// TwinCAT 3 PLC project MotionDevicesPackage
// ProgramVersion: 3.1.4023.0
// libraries:
//   Tc2_MC2, * (Beckhoff Automation GmbH)
//   Tc2_Standard, * (Beckhoff Automation GmbH)
//   Tc2_System, * (Beckhoff Automation GmbH)
//   Tc3_Module, * (Beckhoff Automation GmbH)
// project tree:
//   DUTs/Conveyors/ Conveyor.TcPOU (not stored), ConveyorLSC.TcPOU, ConveyorMode.TcDUT, ConveyorSC.TcPOU, ConveyorSC_NC.TcPOU
//   DUTs/Insertion Package/Drives/ AirPiston.TcPOU, ClearLinkMC.TcPOU, ServoNC.TcPOU, SimplePiston.TcPOU
//   DUTs/Insertion Package/ Homing.TcDUT, Insertion.TcPOU, SuctionPad.TcDUT (not stored)
//   DUTs/Insertion Package/Prototypes/ FBA_Drive.TcPOU, FBA_TrifectaDrive.TcPOU, I_ContinuousDrive.TcIO, I_Drive.TcIO, I_EncodedDrive.TcIO, I_PositionalDrive.TcIO
//   / PlcTask3.TcTTO
//   POUs/ MAIN.TcPOU, WithinTolerance.TcPOU
// (motion and I/O tree: see PLC project conveyorslinking)
// real-time tasks:
//   TASK PlcTask: cycle T#10ms, priority 20, ADS port 350
//   TASK PlcTask1: cycle T#10ms, priority 21, ADS port 351
//   TASK PlcTask2: cycle T#10ms, priority 22, ADS port 352
//   TASK PlcTask3: cycle T#10ms, priority 23, ADS port 353

CONFIGURATION MotionDevicesPackage
    RESOURCE PLC ON TwinCAT3
        TASK PlcTask3(INTERVAL := T#10ms, PRIORITY := 23);
        PROGRAM MAIN WITH PlcTask3 : MAIN;
    END_RESOURCE
END_CONFIGURATION

// ---- DUTs/Conveyors/ConveyorMode.TcDUT
{attribute 'qualified_only'}
//{attribute 'strict'}
TYPE ConveyorMode :
(
	IDLE,
	FORWARD,
	BACKWARD,
	STOP,
	
	size
);
END_TYPE

// ---- DUTs/Insertion Package/Homing.TcDUT
{attribute 'qualified_only'}
{attribute 'strict'}
TYPE Homing :
(
	IDLE,
	
	START,
	RETRY,
	
	STOP,
	SET,
	DONE,
	
	size
);
END_TYPE
(*
general homing sequence:
	on drive.homingSequence() call, home towards home sensor
	if home reached, set position and finish homing as usual
	if outer limit reached, traverse towards inner limit
		when inner limit reached, retry homing
*)

// ---- DUTs/Insertion Package/Prototypes/I_ContinuousDrive.TcIO
INTERFACE I_ContinuousDrive EXTENDS I_Drive

METHOD ABSTRACT moveContinuous : BOOL
VAR_INPUT
	direction : MC_Direction;
END_VAR
END_METHOD

END_INTERFACE

// ---- DUTs/Insertion Package/Prototypes/I_Drive.TcIO
INTERFACE I_Drive

{attribute 'monitoring':='call'}
PROPERTY Active : BOOL
GET
END_GET
END_PROPERTY

{attribute 'monitoring':='call'}
PROPERTY AtHome : BOOL
GET
END_GET
END_PROPERTY

{attribute 'monitoring':='call'}
PROPERTY Error : BOOL
GET
END_GET
END_PROPERTY

{attribute 'monitoring':='call'}
PROPERTY HomeSet : BOOL
GET
END_GET
END_PROPERTY

METHOD ABSTRACT homingSequence : BOOL
VAR_INPUT
END_VAR
END_METHOD

METHOD reset : BOOL
VAR_INPUT
END_VAR
END_METHOD

METHOD ABSTRACT stop : BOOL
VAR_INPUT
END_VAR
END_METHOD

METHOD toHome : BOOL
VAR_INPUT
END_VAR
END_METHOD

END_INTERFACE

// ---- DUTs/Insertion Package/Prototypes/I_EncodedDrive.TcIO
INTERFACE I_EncodedDrive EXTENDS I_PositionalDrive, I_ContinuousDrive
//this drive can perform absolute/relative targeting and continuous motion
//only used if a drive with both encoded and continuous behavior is needed

END_INTERFACE

// ---- DUTs/Insertion Package/Prototypes/I_PositionalDrive.TcIO
INTERFACE I_PositionalDrive EXTENDS I_Drive

PROPERTY CurrentPosition : LREAL
GET
END_GET
SET
END_SET
END_PROPERTY

METHOD ABSTRACT moveAbsolute : BOOL
VAR_INPUT
	newTarget : LREAL; 
END_VAR
END_METHOD

METHOD ABSTRACT moveRelative : BOOL
VAR_INPUT
	distance : LREAL;
END_VAR
END_METHOD

PROPERTY TargetPosition : LREAL
GET
END_GET
SET
END_SET
END_PROPERTY

END_INTERFACE

// ---- POUs/MAIN.TcPOU
PROGRAM MAIN
VAR
	xInsertion : Insertion;
	
	xServoNC : ServoNC;
	xClearLinkMC : ClearLinkMC;
	xAirPiston : AirPiston;
	xSimplePiston : SimplePiston;
	
	xConveyorSC : ConveyorSC;
	xConveyorLSC : ConveyorLSC;
	xConveyorSC_NC : ConveyorSC_NC;
END_VAR

(*
this solution contains the package for various motion devices and the inheritance hierarchy, and any additional types
the Insertion Package folder under DUTs + WithinTolerance() can be copied to any project/module as needed

I_Drive contains the minimum behavior for any drive
FBA_Drive implements I_Drive with the minimum declaration
	FBA_TrifectaDrive extends it by adding an outer limit sensor for drives requiring 3 sensors
	
all Insertion-capable drives extend FBA_Drive or FBA_TrifectaDrive and implement I_ContinuousDrive, I_PositionalDrive, or I_EncodedDrive
*)

END_PROGRAM

// ---- DUTs/Insertion Package/Insertion.TcPOU
FUNCTION_BLOCK Insertion //2d insertion that combines a slider (alignment) and screw (push)
VAR_INPUT //interface references to existing drives
	slider : I_PositionalDrive;
	screw : I_ContinuousDrive;
END_VAR
VAR_OUTPUT
	contact AT %I* : BOOL;
	
	active : BOOL;
	error : BOOL;
	home : BOOL;
	
	homingComplete : BOOL;
	
	sliderPos : LREAL;
END_VAR
(*
this FB encapsulates 2 drives into a generic insertion machine
both drives should be declared externally in Hardware GVL as a concrete FB
Insertion instance should be declared and called in module scope, with the drives from Hardware GVL passed in by Interface reference
*)

homingComplete := slider.HomeSet AND screw.HomeSet;

active := slider.Active OR screw.Active;
error := slider.Error OR screw.Error;
home := slider.AtHome AND screw.AtHome;

sliderPos := slider.CurrentPosition;

METHOD align : BOOL
VAR_INPUT
	targetPos : REAL;
END_VAR
slider.moveAbsolute(newTarget := targetPos);
END_METHOD

METHOD homingSequence : BOOL
VAR_INPUT
END_VAR
IF NOT slider.homeSet THEN
	slider.homingSequence();
END_IF

IF NOT screw.homeSet THEN
	screw.homingSequence();
END_IF

homingSequence := homingComplete;
END_METHOD

METHOD press : BOOL
VAR_INPUT
END_VAR
IF NOT contact THEN
	screw.moveContinuous(direction := MC_Negative_Direction);
END_IF
END_METHOD

METHOD release : BOOL
VAR_INPUT
END_VAR
screw.moveContinuous(direction := MC_Positive_Direction);
END_METHOD

METHOD reset : BOOL
VAR_INPUT
END_VAR
slider.reset();
screw.reset();
END_METHOD

METHOD stop : BOOL
VAR_INPUT
END_VAR
screw.stop();
slider.stop();
END_METHOD

METHOD toHome : BOOL
VAR_INPUT
END_VAR
slider.toHome();
screw.toHome();

toHome := slider.AtHome AND screw.AtHome;
END_METHOD

END_FUNCTION_BLOCK

// ---- DUTs/Insertion Package/Drives/ServoNC.TcPOU
FUNCTION_BLOCK ServoNC EXTENDS FBA_TrifectaDrive IMPLEMENTS I_EncodedDrive
VAR_OUTPUT	
	ready : BOOL;
	position : LREAL;
	velocity : LREAL;
END_VAR
VAR
	axis : AXIS_REF;
	
	mcReadPosition : MC_ReadActualPosition; //continuous enable FBs
	mcReadVelocity : MC_ReadActualVelocity;
	mcReadError : MC_ReadAxisError;
	mcPower : MC_Power;
	
	mcReset : MC_Reset; //rising edge FBs
	mcMoveAbsolute : MC_MoveAbsolute;
	mcMoveRelative : MC_MoveRelative;
	mcMoveVelocity : MC_MoveVelocity;
	
	mcSetPosition : MC_SetPosition;
	mcStop : MC_Stop;
END_VAR
VAR_STAT CONSTANT
	targetingVelocity : INT := 500;
	continuousVelocity : INT := 100;
END_VAR

override();

blocks();

mcReset.Execute := FALSE;
mcMoveAbsolute.Execute := FALSE;
mcMoveRelative.Execute := FALSE;
mcMoveVelocity.Execute := FALSE;
mcSetPosition.Execute := FALSE;
mcStop.Execute := FALSE;

blocks();

ready := bEnable AND NOT Active AND HomeSet;

PROPERTY Active : BOOL
GET
Active := 
	mcMoveAbsolute.Busy OR 
	mcMoveRelative.Busy OR 
	mcMoveVelocity.Busy OR 
	mcSetPosition.Busy OR 
	mcReset.Busy OR 
	mcStop.Busy OR 
	step <> 0;
END_GET
END_PROPERTY

METHOD PRIVATE blocks : BOOL
mcReadPosition(
	Axis:= axis, 
	Enable:= TRUE, 
	Valid=> , 
	Busy=> , 
	Error=> , 
	ErrorID=> , 
	Position=> position);
	
mcReadVelocity(
	Axis:= axis, 
	Enable:= TRUE, 
	Valid=> , 
	Busy=> , 
	Error=> , 
	ErrorID=> , 
	ActualVelocity=> velocity);
	
mcReadError(
	Axis:= axis, 
	Enable:= TRUE, 
	Valid=> , 
	Busy=> , 
	Error=> , 
	ErrorID=> , 
	AxisErrorID=> );

mcReset(
	Axis:= axis, 
	Execute:= , 
	Done=> , 
	Busy=> , 
	Error=> , 
	ErrorID=> );

mcPower(
	Axis:= axis, 
	Enable:= bEnable, 
	Enable_Positive:= TRUE, 
	Enable_Negative:= TRUE, 
	Override:= 100, 
	BufferMode:= , 
	Options:= , 
	Status=> , 
	Busy=> , 
	Active=> , 
	Error=> , 
	ErrorID=> );

mcMoveAbsolute(
	Axis:= axis, 
	Execute:= , 
	Position:= , 
	Velocity:= targetingVelocity, 
	Acceleration:= , 
	Deceleration:= , 
	Jerk:= , 
	BufferMode:= , 
	Options:= , 
	Done=> , 
	Busy=> , 
	Active=> , 
	CommandAborted=> , 
	Error=> , 
	ErrorID=> );
	
mcMoveRelative(
	Axis:= axis, 
	Execute:= , 
	Distance:= ,
	Velocity:= targetingVelocity, 
	Acceleration:= , 
	Deceleration:= , 
	Jerk:= , 
	BufferMode:= , 
	Options:= , 
	Done=> , 
	Busy=> , 
	Active=> , 
	CommandAborted=> , 
	Error=> , 
	ErrorID=> );
	
mcMoveVelocity( //stopped with stop();
	Axis:= axis, 
	Execute:= , 
	Velocity:= continuousVelocity, 
	Acceleration:= , 
	Deceleration:= , 
	Jerk:= , 
	Direction:= , 
	BufferMode:= , 
	Options:= , 
	InVelocity=> , 
	Busy=> , 
	Active=> , 
	CommandAborted=> , 
	Error=> , 
	ErrorID=> );
	
mcSetPosition(
	Axis:= axis, 
	Execute:= , 
	Position:= , 
	Mode:= , 
	Options:= , 
	Done=> , 
	Busy=> , 
	Error=> , 
	ErrorID=> );
	
mcStop(
	Axis:= axis, 
	Execute:= , 
	Deceleration:= , 
	Jerk:= , 
	Options:= , 
	Done=> , 
	Busy=> , 
	Active=> , 
	CommandAborted=> , 
	Error=> , 
	ErrorID=> );
END_METHOD

PROPERTY CurrentPosition : LREAL
GET
CurrentPosition := position;
END_GET
SET
position := CurrentPosition;
END_SET
END_PROPERTY

PROPERTY Error : BOOL
GET
error := 
	mcMoveAbsolute.Error OR 
	mcMoveRelative.Error OR 
	mcMoveVelocity.Error OR 
	mcSetPosition.Error OR 
	mcReset.Error OR 
	mcStop.Error OR
	mcReadError.AxisErrorID > 0;
END_GET
END_PROPERTY

METHOD homingSequence : BOOL
CASE step OF
	Homing.IDLE:
		reset();
		IF bEnable THEN
			step := Homing.START;
		END_IF
		
	Homing.START:
		IF AtHome THEN
			mcMoveVelocity.Execute := FALSE;
			step := Homing.STOP;
			
		ELSIF AtInnerLimit THEN
			mcMoveVelocity.Execute := FALSE;
			step := Homing.RETRY;
			
		ELSE
			mcMoveVelocity.Direction := MC_Negative_Direction;
			mcMoveVelocity.Execute := NOT mcMoveVelocity.Execute;
		END_IF
		
	Homing.RETRY:
		IF AtOuterLimit THEN
			mcMoveVelocity.Execute := FALSE;
			step := Homing.START;
		ELSE
			mcMoveVelocity.Direction := MC_Positive_Direction;
			mcMoveVelocity.Execute := NOT mcMoveVelocity.Execute;
		END_IF
		
	Homing.STOP:
		IF velocity = 0 THEN
			mcStop.Execute := FALSE;
			step := Homing.SET;
		ELSE
			mcStop.Execute := TRUE;
		END_IF
		
	Homing.SET:
		IF position = 0 THEN
			mcSetPosition.Execute := FALSE;
			homingSequence := TRUE;
			step := Homing.DONE;
		ELSE
			mcSetPosition.Position := 0;
			mcSetPosition.Execute := TRUE;
		END_IF
		
	Homing.DONE:
		homingComplete := TRUE;
		step := Homing.IDLE;
		
END_CASE
END_METHOD

METHOD moveAbsolute : BOOL
VAR_INPUT
	newTarget : LREAL;
END_VAR
(*
VAR_OUTPUT
	fault : BOOL;
END_VAR
*)
IF NOT Active AND NOT error THEN
	mcMoveAbsolute.Position := newTarget;
	mcMoveAbsolute.Execute := TRUE;
END_IF

moveAbsolute := (*mcMoveAbsolute.Done AND mcMoveAbsolute.Active;*)
	position = newTarget;
END_METHOD

METHOD moveContinuous : BOOL
VAR_INPUT
	//direction : BOOL; //direction (F = inwards, T = outwards)
	direction : MC_Direction;
END_VAR
(*
IF mcMoveVelocity.Active THEN
	stop();
END_IF

IF NOT mcStop.Done THEN
	RETURN;
END_IF
*)
(*
IF direction THEN
	mcMoveVelocity.Direction := MC_Positive_Direction;
ELSE
	mcMoveVelocity.Direction := MC_Negative_Direction;
END_IF
*)
mcMoveVelocity.Direction := direction;

IF NOT mcMoveVelocity.Error THEN
	mcMoveVelocity.Execute := TRUE;
	moveContinuous := TRUE;
END_IF
END_METHOD

METHOD moveRelative : BOOL
VAR_INPUT
	distance : LREAL;
END_VAR
mcMoveRelative.Distance := distance;

moveRelative := mcMoveRelative.Done;
END_METHOD

METHOD PRIVATE override : BOOL
VAR_INPUT
END_VAR
(*
-at home and attempting to traverse outward
-at outer limit and attempting to traverse outward
-at inner limit and attempting to traverse inwards
*)
(*
inward = negative direction, negative velocity
outward = positive direction, positive velocity
*)

IF error THEN
	stop();
	reset();
	
ELSIF
	AtHome AND (TargetPosition > CurrentPosition OR velocity > 0) OR
	AtInnerLimit AND (TargetPosition > CurrentPosition OR velocity > 0) OR
	AtOuterLimit AND (TargetPosition < CurrentPosition OR velocity < 0)
THEN
	stop();
END_IF
END_METHOD

METHOD reset : BOOL
VAR_INPUT
END_VAR
mcReset.Execute := TRUE;

reset := mcReset.Done;
END_METHOD

METHOD stop : BOOL
VAR_INPUT
END_VAR
mcStop.Execute := TRUE;

mcMoveAbsolute.Execute := FALSE;
mcMoveRelative.Execute := FALSE;
mcMoveVelocity.Execute := FALSE;
END_METHOD

PROPERTY TargetPosition : LREAL
GET
END_GET
SET
moveAbsolute(newTarget := TargetPosition);
END_SET
END_PROPERTY

METHOD toHome : BOOL
VAR_INPUT
END_VAR
moveAbsolute(newTarget := 0);

toHome := AtHome;
END_METHOD

END_FUNCTION_BLOCK

// ---- DUTs/Insertion Package/Prototypes/FBA_TrifectaDrive.TcPOU
FUNCTION_BLOCK ABSTRACT FBA_TrifectaDrive EXTENDS FBA_Drive
VAR
	outerLimit AT %I* : BOOL;
END_VAR
(*
this abstract FB adds a rear limit sensor to FBA_Drive
*)

{attribute 'monitoring':='call'}
PROPERTY AtOuterLimit : BOOL
GET
AtOuterLimit := outerLimit <> limitSensorDefaultState;
END_GET
END_PROPERTY

END_FUNCTION_BLOCK

// ---- DUTs/Insertion Package/Prototypes/FBA_Drive.TcPOU
FUNCTION_BLOCK ABSTRACT FBA_Drive IMPLEMENTS I_Drive
VAR_INPUT
	bEnable : BOOL;
END_VAR
VAR //constructor
	limitSensorDefaultState : BOOL;
	//when a traverse sensor is opposite of this value, the respective property becomes TRUE
	//all sensors for a drive should be of the same type - do not mix & match PNP and NPN sensors on the same drive
END_VAR
VAR		
	homingComplete : BOOL;
	step : Homing;
	
	innerLimit AT %I* : BOOL; //replacable with homeLimit
	home AT %I* : BOOL;
	//not all drives have a rear limit, drives that do must extend from FBA_TrifectaDrive
END_VAR
(*
this abstract FB only specifies the minimum data for any drive
*)

{attribute 'monitoring':='call'}
PROPERTY ABSTRACT Active : BOOL
GET
END_GET
END_PROPERTY

{attribute 'monitoring':='call'}
PROPERTY AtHome : BOOL
GET
AtHome := home <> limitSensorDefaultState;
END_GET
END_PROPERTY

{attribute 'monitoring':='call'}
PROPERTY AtInnerLimit : BOOL
GET
AtInnerLimit := innerLimit <> limitSensorDefaultState;
END_GET
END_PROPERTY

{attribute 'monitoring':='call'}
PROPERTY ABSTRACT Error : BOOL
GET
END_GET
END_PROPERTY

{attribute 'monitoring':='call'}
PROPERTY HomeSet : BOOL
GET
HomeSet := homingComplete;
END_GET
END_PROPERTY

{attribute 'TcRpcEnable'}
METHOD ABSTRACT homingSequence : BOOL
VAR_INPUT
END_VAR
END_METHOD

{attribute 'TcRpcEnable'}
METHOD ABSTRACT reset : BOOL
VAR_INPUT
END_VAR
END_METHOD

{attribute 'TcRpcEnable'}
METHOD ABSTRACT stop : BOOL
VAR_INPUT
END_VAR
END_METHOD

METHOD ABSTRACT toHome : BOOL
VAR_INPUT
END_VAR
END_METHOD

END_FUNCTION_BLOCK

// ---- DUTs/Insertion Package/Drives/ClearLinkMC.TcPOU
FUNCTION_BLOCK ClearLinkMC EXTENDS FBA_TrifectaDrive IMPLEMENTS I_EncodedDrive
VAR_OUTPUT
	pulse AT %Q* : INT;
	brakeRelease AT %Q* : BOOL := TRUE;
	enable : BOOL;
	A : BOOL;
	B : BOOL;
	clear : BOOL;
END_VAR
VAR	
	hlfb AT %I* : REAL := -9999; //high level feedback, if -9999 then servo is idle
	
	outputRegister AT %Q* : INT;
	pulseRequest : INT;
	
	homingDelay : TON;
	resetPulse : TP;
	
	mode : (HOLD, TARGET, CONTINUOUS, RESET_ERR);
	calculation : (IDLE, DOWN, UP, CALCULATE, DONE);
	maxPosition : LREAL;
	
	position, targetPos : LREAL;
	
	pulsePosition : INT;
	pulseCounter : INT;
	rotationsPerPulse : INT; //revolutions per pulse
	displacementPerPulse : LREAL; //displacement per pulse
END_VAR
VAR_STAT CONSTANT
	resetWidth : TIME := T#500MS;
	delayWidth : TIME := T#500MS;
END_VAR
VAR //constructor
	homingDirectionOut : BOOL; 			//homing direction - see <A>
	minPosition : LREAL;
	displacementPerRotation : LREAL; 	//displacement per revolution	
	unitsPerPulse : INT := 800; 		//800 Teknic units per rotation - default setting is 800 units (1 rotation) per pulse
END_VAR

//M-connector output register
outputRegister.0 := enable AND bEnable; 	//enable
outputRegister.1 := A; 						//direction bit - T = outwards, F = inwards
outputRegister.2 := B; 						//homing bit - after startup, set to TRUE to begin homing, then set to FALSE to finish homing
outputRegister.3 := clear; 					//reset bit

rotationsPerPulse := unitsPerPulse/800; //Teknic constant - 800 units per rotation
displacementPerPulse := displacementPerRotation * rotationsPerPulse;

resetPulse(IN:= , PT:= resetWidth, Q=> clear, ET=> ); //reset pulse

IF NOT enable AND NOT AtInnerLimit THEN
	homingComplete := FALSE;
	step := Homing.IDLE;
	mode := HOLD;
END_IF

override();

CASE mode OF		
	HOLD: //hold current position, no motion
		pulse := 0;
		pulseRequest := 0;
	
	TARGET:	//target a given position
		
		IF WithinTolerance(position, targetPos, displacementPerPulse) THEN
			pulseRequest := 0;
			pulse := 0;
			mode := HOLD;
			
		ELSIF NOT Active THEN
			A :=  position < targetPos;
			(*
			2 options to traverse to a target position:
				a)  send all pulses at once - continuous motion but may exceed limits, check for bounds before setting
				b)  1 pulse at a time - choppy but safer
			*)
			targetPos := MAX(targetPos, minPosition); //if below minPosition, set to minPosition
			targetPos := MIN(targetPos, maxPosition); //if above maxPosition, set to maxPosition
			
			pulseRequest := TO_INT(ABS(position - targetPos)/displacementPerPulse);
			//pulseRequest := 1;
		END_IF
		
	CONTINUOUS: //single pulses in the direction specified by moveContinuous()
		pulseRequest := 1;
		
	RESET_ERR: //reset pulse, servo may need to be rehomed aftewards
		pulse := 0;
		pulseRequest := 0;
		resetPulse.IN := TRUE;
		
		IF resetPulse.Q THEN
			resetPulse.IN := FALSE;
			mode := HOLD;
		END_IF
		
END_CASE

sequence();

PROPERTY Active : BOOL
GET
Active := hlfb <> -9999;
END_GET
END_PROPERTY

{attribute 'monitoring':='call'}
PROPERTY AtOuterLimit : BOOL
GET
AtOuterLimit := outerLimit <> limitSensorDefaultState;
END_GET
END_PROPERTY

METHOD PRIVATE calculatePositions : BOOL
(*
the purpose of this method is calculate the position at the outer limit

complete a full range traverse while counting the pulses, then multiply
	displacement per rotation
	rotations per pulse
	number of pulses for the traversal
and add to position at inner limit to get position at outer limit
*)
CASE calculation OF
	IDLE:
		calculation := DOWN;
		
	DOWN:
		moveContinuous(direction := MC_Negative_Direction);
		IF AtInnerLimit THEN
			calculation := UP;
			pulseCounter := 0;
		END_IF
		
	UP:
		moveContinuous(direction := MC_Positive_Direction);
		IF AtHome THEN
			maxPosition := minPosition + (displacementPerRotation * rotationsPerPulse * pulseCounter);
			calculation := DONE;
		END_IF
		
	DONE:
		calculation := 0;
		calculatePositions := TRUE;
		
END_CASE
END_METHOD

PROPERTY CurrentPosition : LREAL
GET
CurrentPosition := position;

//CurrentPosition := pulsePosition * displacementPerPulse;
END_GET
SET
position := CurrentPosition;
END_SET
END_PROPERTY

PROPERTY Error : BOOL
GET
END_GET
END_PROPERTY

METHOD homingSequence : BOOL
homingDelay(IN:= , PT:= delayWidth, Q=> , ET=> );

CASE step OF
	Homing.IDLE:
		enable := TRUE;
		A := FALSE;
		B := TRUE;
		brakeRelease := TRUE;
		
		homingComplete := FALSE;
		
		homingDelay.IN := TRUE;
		IF homingDelay.Q THEN
			homingDelay.IN := FALSE;
			//step := Homing.START;
			step := Homing.RETRY;
		END_IF
		
	Homing.START:
		IF homingDelay.Q THEN
			homingDelay.IN := FALSE;
			step := Homing.SET;
			
		ELSIF AtHome THEN
			homingDelay.IN := TRUE;
			
		ELSIF AtOuterLimit THEN
			step := Homing.RETRY;
		
		ELSE
			enable := TRUE;
			A := FALSE;
			B := TRUE;
			brakeRelease := TRUE;
		
		END_IF
	
	Homing.RETRY:
		IF AtInnerLimit THEN
			homingDelay.IN := TRUE;
			enable := FALSE;
			
			IF homingDelay.Q THEN
				homingDelay.IN := FALSE;
				step := Homing.START;
			END_IF
			
		ELSE
			enable := TRUE;
			A := FALSE;
			B := FALSE;
			brakeRelease := TRUE;
			
			mode := CONTINUOUS;
		END_IF

	Homing.SET:
		enable := TRUE;
		A := FALSE;
		B := FALSE;
		brakeRelease := TRUE;
		
		IF calculatePositions() THEN
			step := Homing.DONE;
		END_IF
		
	Homing.DONE:
		homingSequence := homingComplete := TRUE;
		
		pulsePosition := 0;
		
		mode := HOLD;
		step := Homing.IDLE;
	
END_CASE
END_METHOD

{attribute 'TcRpcEnable'}
METHOD moveAbsolute : BOOL
VAR_INPUT
	newTarget : LREAL;
END_VAR
IF target >= maxPosition AND target <= minPosition THEN
	A :=  position < targetPos;
	targetPos := newTarget;
	mode := TARGET;
	
	moveAbsolute := TRUE;
END_IF
END_METHOD

{attribute 'TcRpcEnable'}
METHOD moveContinuous : BOOL
VAR_INPUT
	direction : MC_Direction;
END_VAR
IF direction = MC_Negative_Direction THEN
	A := FALSE;
ELSIF direction = MC_Positive_Direction THEN
	A := TRUE;
END_IF

mode := CONTINUOUS;
END_METHOD

{attribute 'TcRpcEnable'}
METHOD moveRelative : BOOL
VAR_INPUT
	distance : LREAL;
END_VAR
targetPos := targetPos + distance;

mode := TARGET;
END_METHOD

METHOD PRIVATE override : BOOL
VAR_INPUT
END_VAR
(*
allowable motion is between AtHome and AtInnerLimit
*)
IF AtHome AND NOT Active THEN
	IF homingDirectionOut THEN //homing is outwards
		position := maxPosition;
		pulsePosition := pulseCounter;
	ELSE
		position := minPosition;
		pulsePosition := 0;
	END_IF
	

ELSIF AtInnerLimit AND NOT Active THEN
	IF homingDirectionOut THEN //homing is outwards
		position := minPosition;
		pulsePosition := 0;
	ELSE
		position := maxPosition;
		pulsePosition := pulseCounter;
	END_IF
END_IF

CASE mode OF		
	HOLD:
		//
	
	TARGET:
		IF
			(AtHome AND TargetPosition > CurrentPosition) OR
			(AtInnerLimit AND TargetPosition > CurrentPosition) OR
			(AtOuterLimit AND TargetPosition < CurrentPosition)
		THEN
			mode := HOLD;
		END_IF
		
	CONTINUOUS:
		IF
			(AtHome AND A) OR
			(AtInnerLimit AND A) OR
			(AtOuterLimit AND NOT A)
		THEN
			mode := HOLD;
		END_IF
		
	RESET_ERR:
		//
		
END_CASE
END_METHOD

METHOD reset : BOOL
VAR_INPUT
END_VAR
mode := RESET_ERR;
END_METHOD

METHOD PRIVATE sequence : BOOL
VAR_INPUT
END_VAR
IF Active THEN //servo is active
	IF A THEN //positive direction
		position := position + (displacementPerPulse * pulse);
		pulsePosition := pulsePosition + pulse;
		
		pulseCounter := pulseCounter + pulse;
	ELSE //negative direction
		position := position - (displacementPerPulse * pulse);
		pulsePosition := pulsePosition - pulse;
		
		pulseCounter := pulseCounter - pulse;
	END_IF
	pulse := 0; //pulses already received, can be set to 0 so position change is not compounded

ELSIF pulse = 0 THEN //servo is not active
	pulse := pulseRequest;
END_IF

pulseRequest := 0; //remove this if not working as intended
END_METHOD

METHOD stop : BOOL
VAR_INPUT
END_VAR
mode := HOLD;
END_METHOD

PROPERTY TargetPosition : LREAL
GET
END_GET
SET
targetPos := TargetPosition;
END_SET
END_PROPERTY

METHOD toHome : BOOL
VAR_INPUT
END_VAR
IF homingDirectionOut THEN
	moveAbsolute(newTarget := maxPosition);
ELSE
	moveAbsolute(newTarget := minPosition);
END_IF
END_METHOD

END_FUNCTION_BLOCK

// ---- POUs/WithinTolerance.TcPOU
FUNCTION WithinTolerance : BOOL
VAR_INPUT
	v1 : LREAL;
	v2 : LREAL;
	tolerance : LREAL;
END_VAR

WithinTolerance := ABS(v1-v2) < tolerance;

END_FUNCTION

// ---- DUTs/Insertion Package/Drives/AirPiston.TcPOU
FUNCTION_BLOCK AirPiston EXTENDS FBA_Drive IMPLEMENTS I_ContinuousDrive
VAR_OUTPUT
	valveExtend AT %Q* : BOOL;
	valveRetract AT %Q* : BOOL;
END_VAR
VAR //constructor
	useBrake : BOOL; //optional - set to FALSE if retraction brake pulse is not required
END_VAR
VAR
	mode : (HOLD, IN, OUT, BRAKE);
	brakePulse : TP; //generates the retraction pulse
END_VAR
VAR_STAT CONSTANT
	brakeWidth : TIME := T#650MS;
END_VAR

IF NOT bEnable THEN
	stop();
	RETURN;
END_IF

brakePulse(IN:= , PT:= brakeWidth, Q=> , ET=> ); //reversal to act as brake
brakePulse.IN := brakePulse.IN AND brakePulse.Q; //automatically turn off pulse

override(); //alters the mode to prevent exceeding limits

CASE mode OF
	HOLD:
		valveExtend := FALSE;
		valveRetract := FALSE;
		
	IN:
		valveExtend := TRUE;
		valveRetract := FALSE;
		
	OUT:
		valveExtend := FALSE;
		valveRetract := TRUE;
		
	BRAKE: //coasts past inner limit, then slides back
		valveExtend := FALSE;
		valveRetract := TRUE;
		
		IF AtHome THEN
			mode := HOLD;
		END_IF
		
END_CASE

valveRetract := valveRetract OR brakePulse.Q; //from mode or brake

PROPERTY Active : BOOL
GET
Active :=
	mode <> HOLD AND
	valveExtend OR valveRetract;
END_GET
END_PROPERTY

PROPERTY Error : BOOL
GET
END_GET
END_PROPERTY

METHOD extend : BOOL
VAR_INPUT
END_VAR
IF mode <> BRAKE THEN
	mode := IN;
END_IF
END_METHOD

METHOD homingSequence : BOOL
CASE step OF
	Homing.IDLE:
		step := Homing.START;
		
	Homing.START:
		IF AtHome THEN //if reached home
			step := Homing.DONE;
		ELSE
			mode := OUT;
		END_IF
		
	Homing.DONE:
		mode := HOLD;
		homingComplete := TRUE;
		homingSequence := TRUE;		
	
END_CASE
END_METHOD

{attribute 'TcRpcEnable'}
METHOD moveContinuous : BOOL
VAR_INPUT
	direction : MC_Direction;
END_VAR
IF direction = MC_Positive_Direction THEN
	retract();
ELSIF direction = MC_Negative_Direction THEN
	extend();
END_IF
END_METHOD

METHOD PRIVATE override : BOOL
VAR_INPUT
END_VAR
IF brakePulse.Q THEN
	mode := HOLD;
END_IF

IF AtHome AND (valveRetract OR mode = OUT) THEN
	mode := HOLD;
	
ELSIF AtInnerLimit AND (valveExtend OR mode = IN) THEN	
	brakePulse.IN := useBrake;
	mode := HOLD;
END_IF


IF NOT bEnable THEN
	stop();
END_IF
END_METHOD

METHOD reset : BOOL
VAR_INPUT
END_VAR
stop();
END_METHOD

METHOD retract : BOOL
VAR_INPUT
END_VAR
IF mode <> BRAKE THEN
	mode := OUT;
END_IF
END_METHOD

METHOD stop : BOOL
VAR_INPUT
END_VAR
valveExtend := FALSE;
valveRetract := FALSE;
mode := HOLD;
END_METHOD

METHOD toHome : BOOL
VAR_INPUT
END_VAR
mode := OUT;
END_METHOD

END_FUNCTION_BLOCK

// ---- DUTs/Insertion Package/Drives/SimplePiston.TcPOU
FUNCTION_BLOCK SimplePiston
VAR_INPUT
	bEnable : BOOL;
END_VAR
VAR_OUTPUT
	pistonExtend AT %Q* : BOOL;
	pistonRetract AT %Q* : BOOL;
	
	extended AT %I* : BOOL;
	retracted AT %I* : BOOL;
	
	busy : BOOL;
END_VAR
VAR
	mode : (HOLD, IN, OUT);
END_VAR

IF
	NOT bEnable OR
	(retracted AND_THEN (pistonRetract OR mode = OUT)) OR
	(extended AND_THEN (pistonExtend OR mode = IN))
THEN
	mode := HOLD;
END_IF

CASE mode OF
	HOLD:
		pistonRetract := FALSE;
		pistonExtend := FALSE;
		
	IN:
		pistonRetract := FALSE;
		pistonExtend := TRUE;
	
	OUT:
		pistonRetract := TRUE;
		pistonExtend := FALSE;
	
END_CASE

busy := mode = IN OR mode = OUT;

METHOD extend : BOOL
VAR_INPUT
END_VAR
mode := IN;
END_METHOD

METHOD retract : BOOL
VAR_INPUT
END_VAR
mode := OUT;

retract := retracted;
END_METHOD

METHOD stop : BOOL
VAR_INPUT
END_VAR
pistonExtend := FALSE;
pistonRetract := FALSE;
mode := HOLD;
END_METHOD

END_FUNCTION_BLOCK

// ---- DUTs/Conveyors/ConveyorSC.TcPOU
FUNCTION_BLOCK ConveyorSC
VAR_INPUT
	bEnable : BOOL;
END_VAR
VAR_OUTPUT
	trueMode : ConveyorMode;
	requestedMode : ConveyorMode;
	
	error AT %I* : BOOL;
	position AT %I* : REAL;
	velocity AT %I* : REAL;
END_VAR
VAR
	enable AT %Q* : BOOL := TRUE;
	direction AT %Q* : BOOL; //FALSE = forward, TRUE = backward
	pulse AT %Q* : BOOL;
	reset AT %Q* : BOOL;
	
	sensorEntry AT %I* : BOOL := TRUE;
	sensorExit AT %I* : BOOL;
END_VAR
VAR
	//nextConveyor : POINTER TO ConveyorSC;
	//prevConveyor : POINTER TO ConveyorSC;
	
	pulser : TP; //pulses are assumed to be low-high-low
END_VAR
VAR_STAT CONSTANT
	pulseWidth : TIME := T#50MS;
END_VAR
(*
standard slat conveyor - no lifter
compliant with PLCopen motion control
*)

enable := bEnable;

override();

sequence();

METHOD backward : BOOL
VAR_INPUT
END_VAR
END_METHOD

METHOD forward : BOOL
VAR_INPUT
END_VAR
END_METHOD

{attribute 'monitoring' := 'call'}
PROPERTY IsOccupied : BOOL
GET
IsOccupied := sensorExit OR sensorEntry;
END_GET
END_PROPERTY

METHOD join : BOOL
VAR_INPUT
	conveyor : POINTER TO ConveyorSC;
END_VAR
//nextConveyor := conveyor;
//conveyor^.prevConveyor := THIS;
END_METHOD

METHOD PROTECTED override : BOOL
VAR_INPUT
END_VAR
END_METHOD

METHOD reset : BOOL
VAR_INPUT
END_VAR
position := 0;
velocity := velocity; //no change
END_METHOD

METHOD PROTECTED sequence : BOOL
VAR_INPUT
END_VAR
direction := (trueMode = ConveyorMode.BACKWARD); //set direction bit

pulser(IN:= , PT:= pulseWidth, Q=> pulse, ET=> );
pulser.IN := 
	enable AND 
	NOT error AND 
	NOT reset AND 
	(trueMode = ConveyorMode.FORWARD OR trueMode = ConveyorMode.BACKWARD)
	AND pulser.Q; //ends pulse itself
END_METHOD

METHOD setMode : BOOL
VAR_INPUT
	mode : ConveyorMode;
END_VAR
trueMode := mode;
END_METHOD

METHOD setRequest : BOOL
VAR_INPUT
	newRequest : ConveyorMode;
END_VAR
requestedMode := newRequest;
END_METHOD

METHOD target : BOOL
VAR_INPUT
	targetPosition : REAL;
END_VAR
END_METHOD

END_FUNCTION_BLOCK

// ---- DUTs/Conveyors/ConveyorLSC.TcPOU
FUNCTION_BLOCK ConveyorLSC EXTENDS ConveyorSC
VAR_OUTPUT
	lifterError AT %I* : BOOL;
	
	extended AT %I* : BOOL;
	retracted AT %I* : BOOL;
END_VAR
VAR	
	lifterEnable AT %Q* : BOOL := TRUE;
	lifterDirection AT %Q* : BOOL; //FALSE = up, TRUE = down
	lifterPulse AT %Q* : BOOL;
	lifterReset AT %Q* : BOOL;
END_VAR
VAR	
	lifterMode : (HOLD, LIFTER_EXTEND, LIFTER_RETRACT); 
	lifterPulser : TP; //pulses are assumed to be low-high-low
END_VAR

SUPER^();

lifterOverride();

lifterSequence();

METHOD backward : BOOL
VAR_INPUT
END_VAR
END_METHOD

METHOD extend : BOOL
VAR_INPUT
END_VAR
lifterMode := LIFTER_EXTEND;
END_METHOD

METHOD forward : BOOL
VAR_INPUT
END_VAR
END_METHOD

METHOD PROTECTED lifterOverride : BOOL
VAR_INPUT
END_VAR
IF
	(extended AND lifterMode = LIFTER_EXTEND) OR
	(retracted AND lifterMode = LIFTER_RETRACT)
THEN
	lifterMode := HOLD;
END_IF
END_METHOD

METHOD PROTECTED lifterSequence : BOOL
VAR_INPUT
END_VAR
VAR
	nextOp, prevOp : INT;
END_VAR
lifterPulser(IN:= , PT:= pulseWidth, Q=> , ET=> );
lifterPulser.IN := 
	lifterEnable AND 
	NOT lifterError AND 
	NOT lifterReset AND 
	( (lifterMode = LIFTER_EXTEND AND NOT extended) OR (lifterMode = LIFTER_RETRACT AND NOT retracted) ) AND
	lifterPulser.Q; //self-ending pulse

lifterPulse := lifterPulser.Q AND lifterPulser.ET < pulseWidth/2;
END_METHOD

METHOD reset : BOOL
VAR_INPUT
END_VAR
position := 0;
velocity := velocity; //no change

extend();
END_METHOD

METHOD retract : BOOL
VAR_INPUT
END_VAR
lifterMode := LIFTER_RETRACT;
END_METHOD

END_FUNCTION_BLOCK

// ---- DUTs/Conveyors/ConveyorSC_NC.TcPOU
FUNCTION_BLOCK ConveyorSC_NC
VAR_INPUT
	bEnable : BOOL;
END_VAR
VAR_OUTPUT
	sensorEntry AT %I* : BOOL := TRUE;
	sensorExit AT %I* : BOOL := TRUE;
	
	trueMode : ConveyorMode;
	requestedMode : ConveyorMode;
	
	position : LREAL;
	velocity : LREAL;
	ready : BOOL;
END_VAR
VAR
	axis : AXIS_REF;
	
	mcReadPosition : MC_ReadActualPosition; //continuous enable FBs
	mcReadVelocity : MC_ReadActualVelocity;
	mcReadError : MC_ReadAxisError;
	mcPower : MC_Power;
	
	mcReset : MC_Reset; //rising edge FBs
	mcMoveAbsolute : MC_MoveAbsolute;
	mcMoveRelative : MC_MoveRelative;
	mcMoveVelocity : MC_MoveVelocity;
	
	mcSetPosition : MC_SetPosition;
	mcStop : MC_Stop;
END_VAR
VAR_STAT CONSTANT
	targetingVelocity : INT := 500;
	continuousVelocity : INT := 500;
END_VAR
(*
this FB represents a standard slat conveyor with no lifter
	compliant with PLCopen motion control

unlike standalone servos,
	conveyors need to coordinate (not slave) their motion with other conveyors
	and be able to set their current position to any value as required by the system
	
moveAbsolute is provided for now but should not be used for position targetting and may be protected/privated later
instead, request/set the operation mode and the motion will follow
*)

IF error THEN
	stop();
	reset();
	
ELSE
	CASE trueMode OF
		ConveyorMode.IDLE:			stop();	
		ConveyorMode.FORWARD:		moveContinuous(direction:= MC_Positive_Direction);
		ConveyorMode.BACKWARD:		moveContinuous(direction:= MC_Negative_Direction);
		ConveyorMode.STOP:			stop();
	END_CASE
	
END_IF

blocks();

mcReset.Execute := FALSE;
mcMoveAbsolute.Execute := FALSE;
mcMoveRelative.Execute := FALSE;
mcMoveVelocity.Execute := FALSE;
mcSetPosition.Execute := FALSE;
mcStop.Execute := FALSE;

blocks();

PROPERTY Active : BOOL
GET
Active := 
	mcMoveAbsolute.Busy OR 
	mcMoveRelative.Busy OR 
	mcMoveVelocity.Busy OR 
	mcSetPosition.Busy OR 
	mcReset.Busy OR 
	mcStop.Busy;
END_GET
END_PROPERTY

METHOD PRIVATE blocks : BOOL
mcReadPosition(
	Axis:= axis, 
	Enable:= TRUE, 
	Valid=> , 
	Busy=> , 
	Error=> , 
	ErrorID=> , 
	Position=> position);
	
mcReadVelocity(
	Axis:= axis, 
	Enable:= TRUE, 
	Valid=> , 
	Busy=> , 
	Error=> , 
	ErrorID=> , 
	ActualVelocity=> velocity);
	
mcReadError(
	Axis:= axis, 
	Enable:= TRUE, 
	Valid=> , 
	Busy=> , 
	Error=> , 
	ErrorID=> , 
	AxisErrorID=> );
	
mcPower(
	Axis:= axis, 
	Enable:= bEnable, 
	Enable_Positive:= TRUE, 
	Enable_Negative:= TRUE, 
	Override:= 100, 
	BufferMode:= , 
	Options:= , 
	Status=> , 
	Busy=> , 
	Active=> , 
	Error=> , 
	ErrorID=> );

mcReset(
	Axis:= axis, 
	Execute:= , 
	Done=> , 
	Busy=> , 
	Error=> , 
	ErrorID=> );

mcMoveAbsolute(
	Axis:= axis, 
	Execute:= , 
	Position:= , 
	Velocity:= targetingVelocity, 
	Acceleration:= , 
	Deceleration:= , 
	Jerk:= , 
	BufferMode:= , 
	Options:= , 
	Done=> , 
	Busy=> , 
	Active=> , 
	CommandAborted=> , 
	Error=> , 
	ErrorID=> );
	
mcMoveRelative(
	Axis:= axis, 
	Execute:= , 
	Distance:= ,
	Velocity:= targetingVelocity, 
	Acceleration:= , 
	Deceleration:= , 
	Jerk:= , 
	BufferMode:= , 
	Options:= , 
	Done=> , 
	Busy=> , 
	Active=> , 
	CommandAborted=> , 
	Error=> , 
	ErrorID=> );
	
mcMoveVelocity( //stopped with stop();
	Axis:= axis, 
	Execute:= , 
	Velocity:= continuousVelocity, 
	Acceleration:= , 
	Deceleration:= , 
	Jerk:= , 
	Direction:= , 
	BufferMode:= , 
	Options:= , 
	InVelocity=> , 
	Busy=> , 
	Active=> , 
	CommandAborted=> , 
	Error=> , 
	ErrorID=> );
	
mcSetPosition(
	Axis:= axis, 
	Execute:= , 
	Position:= , 
	Mode:= , 
	Options:= , 
	Done=> , 
	Busy=> , 
	Error=> , 
	ErrorID=> );
	
mcStop(
	Axis:= axis, 
	Execute:= , 
	Deceleration:= , 
	Jerk:= , 
	Options:= , 
	Done=> , 
	Busy=> , 
	Active=> , 
	CommandAborted=> , 
	Error=> , 
	ErrorID=> );
END_METHOD

PROPERTY CurrentPosition : LREAL
GET
CurrentPosition := position;
END_GET
SET
position := CurrentPosition;
END_SET
END_PROPERTY

PROPERTY Error : BOOL
GET
error := 
	mcMoveAbsolute.Error OR 
	mcMoveRelative.Error OR 
	mcMoveVelocity.Error OR 
	mcSetPosition.Error OR 
	mcReset.Error OR 
	mcStop.Error OR
	mcReadError.AxisErrorID > 0;
END_GET
END_PROPERTY

{attribute 'monitoring' := 'call'}
PROPERTY IsOccupied : BOOL
GET
IsOccupied := sensorExit OR sensorEntry;
END_GET
END_PROPERTY

METHOD moveAbsolute : BOOL
VAR_INPUT
	newTarget : LREAL;
END_VAR
mcMoveAbsolute.Position := newTarget;

IF NOT Active AND NOT error THEN
	mcMoveAbsolute.Execute := TRUE;
END_IF

moveAbsolute := 
	//mcMoveAbsolute.Done;
	CurrentPosition = TargetPosition;
END_METHOD

METHOD moveContinuous : BOOL
VAR_INPUT
	direction : MC_Direction;
END_VAR
mcMoveVelocity.Direction := direction;

IF NOT Active AND NOT error THEN
	mcMoveVelocity.Execute := TRUE;
	moveContinuous := TRUE;
END_IF
END_METHOD

METHOD reset : BOOL
VAR_INPUT
END_VAR
mcReset.Execute := TRUE;

reset := mcReset.Done;
END_METHOD

METHOD setMode : BOOL
VAR_INPUT
	mode : ConveyorMode;
END_VAR
trueMode := mode;
END_METHOD

METHOD setRequest : BOOL
VAR_INPUT
	newRequest : ConveyorMode;
END_VAR
requestedMode := newRequest;
END_METHOD

METHOD stop : BOOL
VAR_INPUT
END_VAR
mcStop.Execute := TRUE;

mcMoveAbsolute.Execute := FALSE;
mcMoveRelative.Execute := FALSE;
mcMoveVelocity.Execute := FALSE;
END_METHOD

PROPERTY TargetPosition : LREAL
GET
END_GET
SET
moveAbsolute(newTarget := TargetPosition);
END_SET
END_PROPERTY

END_FUNCTION_BLOCK
